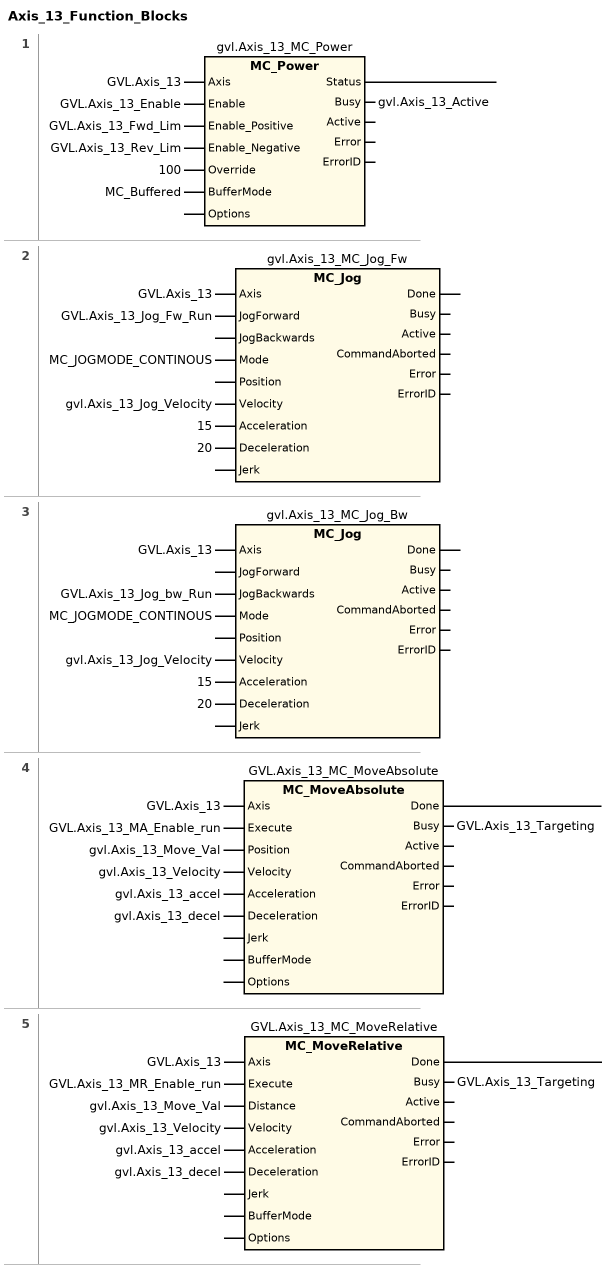
// NETWORK 1
gvl.Axis_13_MC_Power(
    Axis := GVL.Axis_13,
    Enable := GVL.Axis_13_Enable,
    Enable_Positive := GVL.Axis_13_Fwd_Lim,
    Enable_Negative := GVL.Axis_13_Rev_Lim,
    Override := 100,
    BufferMode := MC_Buffered,
    Busy => gvl.Axis_13_Active); // MC_Power

// NETWORK 2
gvl.Axis_13_MC_Jog_Fw(
    Axis := GVL.Axis_13,
    JogForward := GVL.Axis_13_Jog_Fw_Run,
    Mode := MC_JOGMODE_CONTINOUS,
    Velocity := gvl.Axis_13_Jog_Velocity,
    Acceleration := 15,
    Deceleration := 20); // MC_Jog

// NETWORK 3
gvl.Axis_13_MC_Jog_Bw(
    Axis := GVL.Axis_13,
    JogBackwards := GVL.Axis_13_Jog_bw_Run,
    Mode := MC_JOGMODE_CONTINOUS,
    Velocity := gvl.Axis_13_Jog_Velocity,
    Acceleration := 15,
    Deceleration := 20); // MC_Jog

// NETWORK 4
GVL.Axis_13_MC_MoveAbsolute(
    Axis := GVL.Axis_13,
    Execute := GVL.Axis_13_MA_Enable_run,
    Position := gvl.Axis_13_Move_Val,
    Velocity := gvl.Axis_13_Velocity,
    Acceleration := gvl.Axis_13_accel,
    Deceleration := gvl.Axis_13_decel,
    Busy => GVL.Axis_13_Targeting); // MC_MoveAbsolute

// NETWORK 5
GVL.Axis_13_MC_MoveRelative(
    Axis := GVL.Axis_13,
    Execute := GVL.Axis_13_MR_Enable_run,
    Distance := gvl.Axis_13_Move_Val,
    Velocity := gvl.Axis_13_Velocity,
    Acceleration := gvl.Axis_13_accel,
    Deceleration := gvl.Axis_13_decel,
    Busy => GVL.Axis_13_Targeting); // MC_MoveRelative

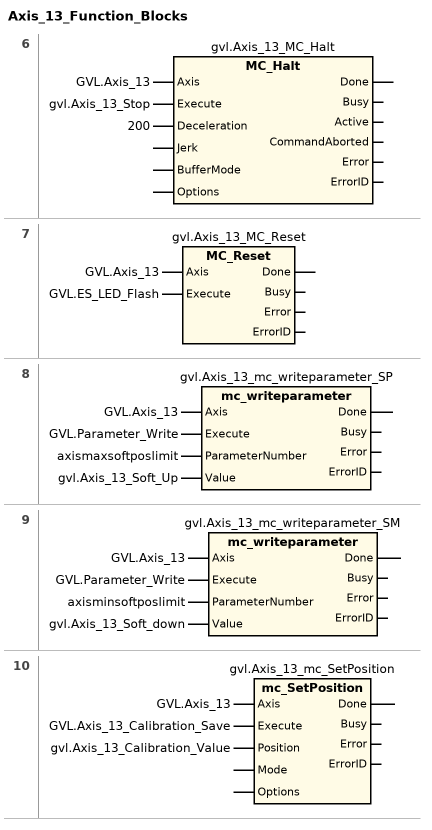
// NETWORK 6
gvl.Axis_13_MC_Halt(Axis := GVL.Axis_13, Execute := gvl.Axis_13_Stop, Deceleration := 200); // MC_Halt

// NETWORK 7
gvl.Axis_13_MC_Reset(Axis := GVL.Axis_13, Execute := GVL.ES_LED_Flash); // MC_Reset

// NETWORK 8
gvl.Axis_13_mc_writeparameter_SP(
    Axis := GVL.Axis_13,
    Execute := GVL.Parameter_Write,
    ParameterNumber := axismaxsoftposlimit,
    Value := gvl.Axis_13_Soft_Up); // mc_writeparameter

// NETWORK 9
gvl.Axis_13_mc_writeparameter_SM(
    Axis := GVL.Axis_13,
    Execute := GVL.Parameter_Write,
    ParameterNumber := axisminsoftposlimit,
    Value := gvl.Axis_13_Soft_down); // mc_writeparameter

// NETWORK 10
gvl.Axis_13_mc_SetPosition(
    Axis := GVL.Axis_13,
    Execute := GVL.Axis_13_Calibration_Save,
    Position := gvl.Axis_13_Calibration_Value); // mc_SetPosition

END_PROGRAM

// ---- POUs/Axis_13_Logic.TcPOU
PROGRAM Axis_13_Logic
VAR
	TON_0: TON;
	TON_1: TON;
	TON_2: TON;
	TON_3: TON;
	Axis_13_Velocity_Range: LREAL;
	Axis_13_Velocity_Scale: LREAL;
	Axis_13_Velocity_Raw: LREAL;
	Axis_13_Soft_Range: LREAL;
	Axis_13_Soft_Position: LREAL;
	Axis_13_Soft_Position_In_Range: LREAL;
END_VAR

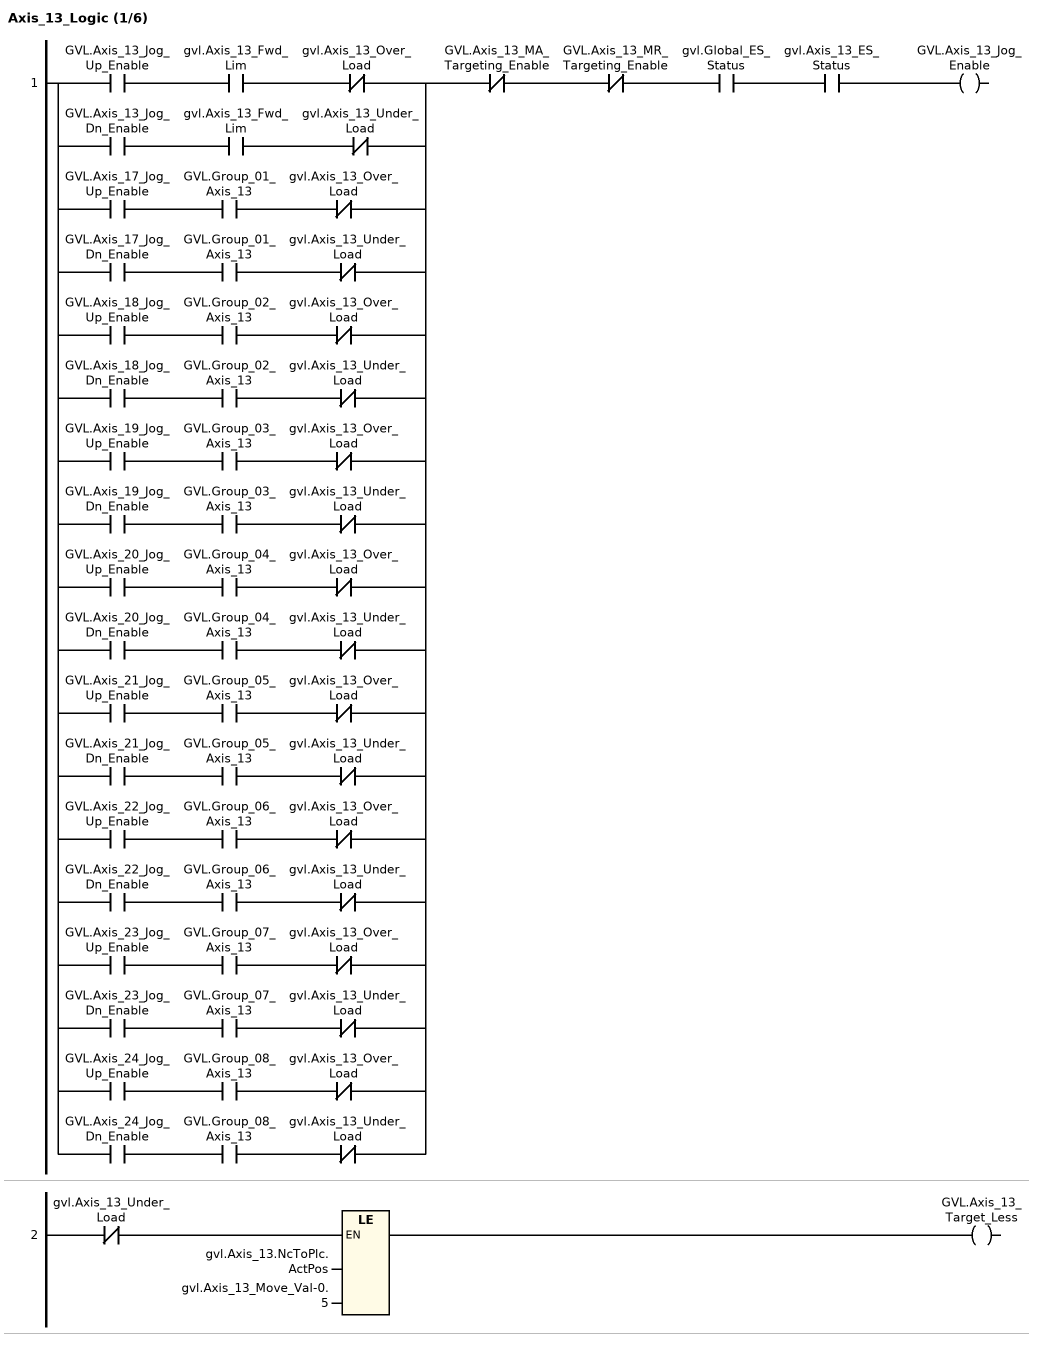
// NETWORK 1
GVL.Axis_13_Jog_Enable := (GVL.Axis_13_Jog_Up_Enable AND gvl.Axis_13_Fwd_Lim AND NOT gvl.Axis_13_Over_Load OR GVL.Axis_13_Jog_Dn_Enable AND gvl.Axis_13_Fwd_Lim AND NOT gvl.Axis_13_Under_Load OR GVL.Axis_17_Jog_Up_Enable AND GVL.Group_01_Axis_13 AND NOT gvl.Axis_13_Over_Load OR GVL.Axis_17_Jog_Dn_Enable AND GVL.Group_01_Axis_13 AND NOT gvl.Axis_13_Under_Load OR GVL.Axis_18_Jog_Up_Enable AND GVL.Group_02_Axis_13 AND NOT gvl.Axis_13_Over_Load OR GVL.Axis_18_Jog_Dn_Enable AND GVL.Group_02_Axis_13 AND NOT gvl.Axis_13_Under_Load OR GVL.Axis_19_Jog_Up_Enable AND GVL.Group_03_Axis_13 AND NOT gvl.Axis_13_Over_Load OR GVL.Axis_19_Jog_Dn_Enable AND GVL.Group_03_Axis_13 AND NOT gvl.Axis_13_Under_Load OR GVL.Axis_20_Jog_Up_Enable AND GVL.Group_04_Axis_13 AND NOT gvl.Axis_13_Over_Load OR GVL.Axis_20_Jog_Dn_Enable AND GVL.Group_04_Axis_13 AND NOT gvl.Axis_13_Under_Load OR GVL.Axis_21_Jog_Up_Enable AND GVL.Group_05_Axis_13 AND NOT gvl.Axis_13_Over_Load OR GVL.Axis_21_Jog_Dn_Enable AND GVL.Group_05_Axis_13 AND NOT gvl.Axis_13_Under_Load OR GVL.Axis_22_Jog_Up_Enable AND GVL.Group_06_Axis_13 AND NOT gvl.Axis_13_Over_Load OR GVL.Axis_22_Jog_Dn_Enable AND GVL.Group_06_Axis_13 AND NOT gvl.Axis_13_Under_Load OR GVL.Axis_23_Jog_Up_Enable AND GVL.Group_07_Axis_13 AND NOT gvl.Axis_13_Over_Load OR GVL.Axis_23_Jog_Dn_Enable AND GVL.Group_07_Axis_13 AND NOT gvl.Axis_13_Under_Load OR GVL.Axis_24_Jog_Up_Enable AND GVL.Group_08_Axis_13 AND NOT gvl.Axis_13_Over_Load OR GVL.Axis_24_Jog_Dn_Enable AND GVL.Group_08_Axis_13 AND NOT gvl.Axis_13_Under_Load) AND NOT GVL.Axis_13_MA_Targeting_Enable AND NOT GVL.Axis_13_MR_Targeting_Enable AND gvl.Global_ES_Status AND gvl.Axis_13_ES_Status;

// NETWORK 2
GVL.Axis_13_Target_Less := NOT gvl.Axis_13_Under_Load AND gvl.Axis_13.NcToPlc.ActPos <= (gvl.Axis_13_Move_Val-0.5);

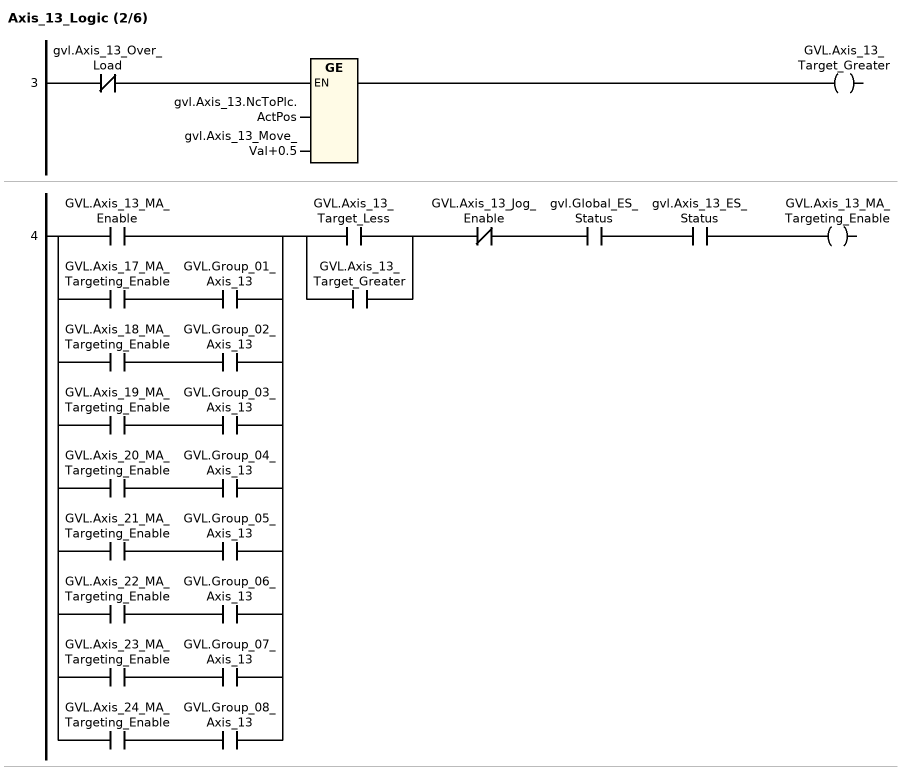
// NETWORK 3
GVL.Axis_13_Target_Greater := NOT gvl.Axis_13_Over_Load AND gvl.Axis_13.NcToPlc.ActPos >= (gvl.Axis_13_Move_Val+0.5);

// NETWORK 4
GVL.Axis_13_MA_Targeting_Enable := (GVL.Axis_13_MA_Enable OR GVL.Axis_17_MA_Targeting_Enable AND GVL.Group_01_Axis_13 OR GVL.Axis_18_MA_Targeting_Enable AND GVL.Group_02_Axis_13 OR GVL.Axis_19_MA_Targeting_Enable AND GVL.Group_03_Axis_13 OR GVL.Axis_20_MA_Targeting_Enable AND GVL.Group_04_Axis_13 OR GVL.Axis_21_MA_Targeting_Enable AND GVL.Group_05_Axis_13 OR GVL.Axis_22_MA_Targeting_Enable AND GVL.Group_06_Axis_13 OR GVL.Axis_23_MA_Targeting_Enable AND GVL.Group_07_Axis_13 OR GVL.Axis_24_MA_Targeting_Enable AND GVL.Group_08_Axis_13) AND (GVL.Axis_13_Target_Less OR GVL.Axis_13_Target_Greater) AND NOT GVL.Axis_13_Jog_Enable AND gvl.Global_ES_Status AND gvl.Axis_13_ES_Status;

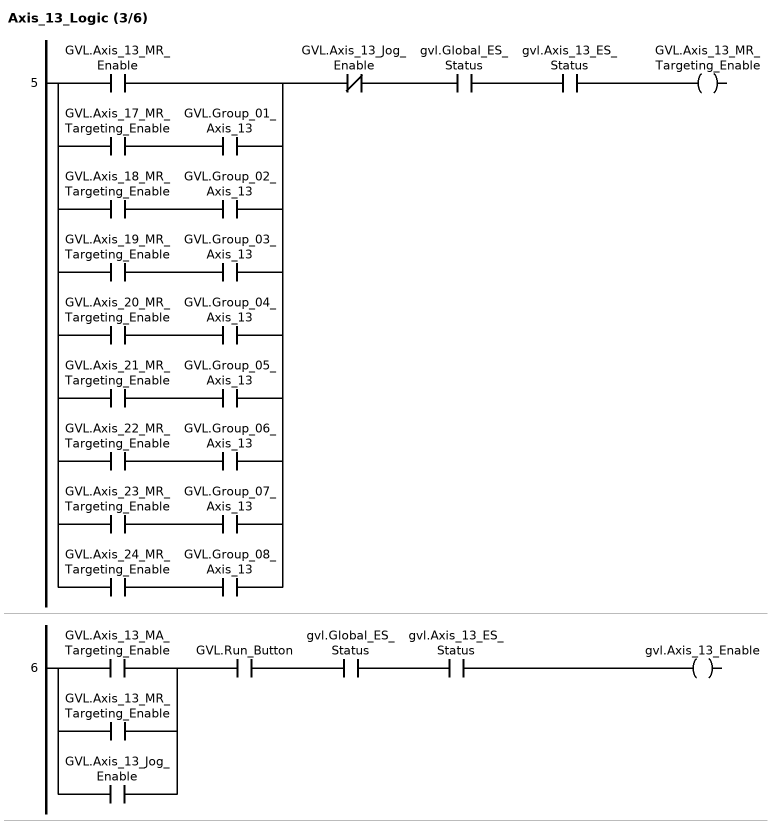
// NETWORK 5
GVL.Axis_13_MR_Targeting_Enable := (GVL.Axis_13_MR_Enable OR GVL.Axis_17_MR_Targeting_Enable AND GVL.Group_01_Axis_13 OR GVL.Axis_18_MR_Targeting_Enable AND GVL.Group_02_Axis_13 OR GVL.Axis_19_MR_Targeting_Enable AND GVL.Group_03_Axis_13 OR GVL.Axis_20_MR_Targeting_Enable AND GVL.Group_04_Axis_13 OR GVL.Axis_21_MR_Targeting_Enable AND GVL.Group_05_Axis_13 OR GVL.Axis_22_MR_Targeting_Enable AND GVL.Group_06_Axis_13 OR GVL.Axis_23_MR_Targeting_Enable AND GVL.Group_07_Axis_13 OR GVL.Axis_24_MR_Targeting_Enable AND GVL.Group_08_Axis_13) AND NOT GVL.Axis_13_Jog_Enable AND gvl.Global_ES_Status AND gvl.Axis_13_ES_Status;

// NETWORK 6
gvl.Axis_13_Enable := (GVL.Axis_13_MA_Targeting_Enable OR GVL.Axis_13_MR_Targeting_Enable OR GVL.Axis_13_Jog_Enable) AND GVL.Run_Button AND gvl.Global_ES_Status AND gvl.Axis_13_ES_Status;

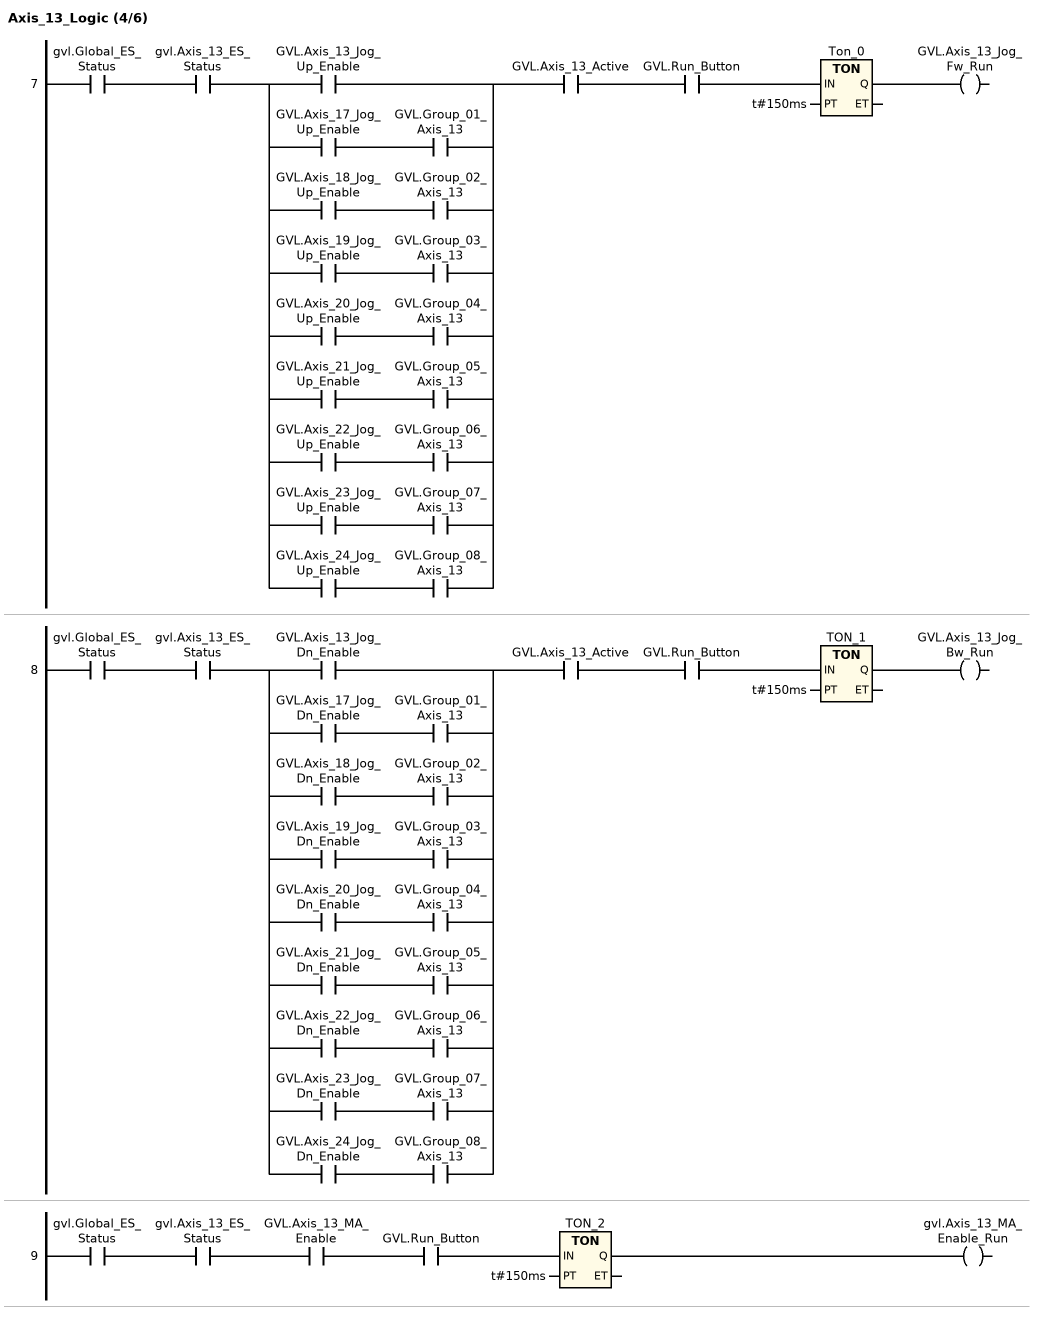
// NETWORK 7
Ton_0(IN := gvl.Global_ES_Status AND gvl.Axis_13_ES_Status AND (GVL.Axis_13_Jog_Up_Enable OR GVL.Axis_17_Jog_Up_Enable AND GVL.Group_01_Axis_13 OR GVL.Axis_18_Jog_Up_Enable AND GVL.Group_02_Axis_13 OR GVL.Axis_19_Jog_Up_Enable AND GVL.Group_03_Axis_13 OR GVL.Axis_20_Jog_Up_Enable AND GVL.Group_04_Axis_13 OR GVL.Axis_21_Jog_Up_Enable AND GVL.Group_05_Axis_13 OR GVL.Axis_22_Jog_Up_Enable AND GVL.Group_06_Axis_13 OR GVL.Axis_23_Jog_Up_Enable AND GVL.Group_07_Axis_13 OR GVL.Axis_24_Jog_Up_Enable AND GVL.Group_08_Axis_13) AND GVL.Axis_13_Active AND GVL.Run_Button, PT := t#150ms); // TON
GVL.Axis_13_Jog_Fw_Run := Ton_0.Q;

// NETWORK 8
TON_1(IN := gvl.Global_ES_Status AND gvl.Axis_13_ES_Status AND (GVL.Axis_13_Jog_Dn_Enable OR GVL.Axis_17_Jog_Dn_Enable AND GVL.Group_01_Axis_13 OR GVL.Axis_18_Jog_Dn_Enable AND GVL.Group_02_Axis_13 OR GVL.Axis_19_Jog_Dn_Enable AND GVL.Group_03_Axis_13 OR GVL.Axis_20_Jog_Dn_Enable AND GVL.Group_04_Axis_13 OR GVL.Axis_21_Jog_Dn_Enable AND GVL.Group_05_Axis_13 OR GVL.Axis_22_Jog_Dn_Enable AND GVL.Group_06_Axis_13 OR GVL.Axis_23_Jog_Dn_Enable AND GVL.Group_07_Axis_13 OR GVL.Axis_24_Jog_Dn_Enable AND GVL.Group_08_Axis_13) AND GVL.Axis_13_Active AND GVL.Run_Button, PT := t#150ms); // TON
GVL.Axis_13_Jog_Bw_Run := TON_1.Q;

// NETWORK 9
TON_2(IN := gvl.Global_ES_Status AND gvl.Axis_13_ES_Status AND GVL.Axis_13_MA_Enable AND GVL.Run_Button, PT := t#150ms); // TON
gvl.Axis_13_MA_Enable_Run := TON_2.Q;

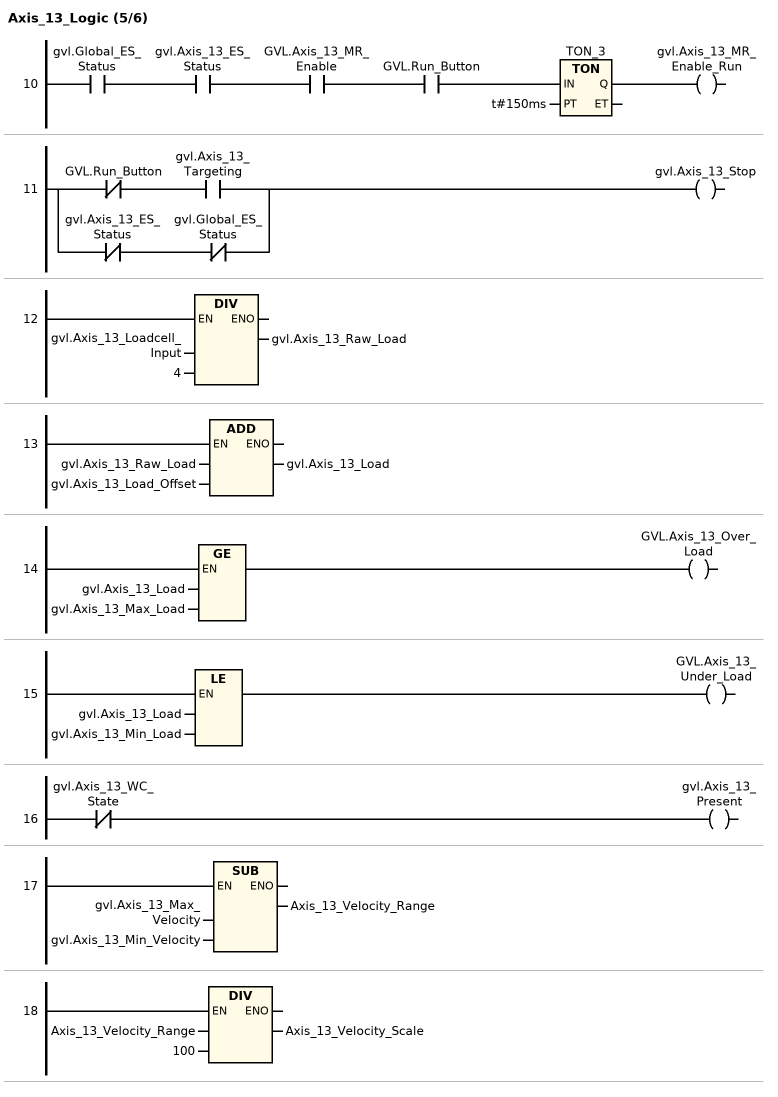
// NETWORK 10
TON_3(IN := gvl.Global_ES_Status AND gvl.Axis_13_ES_Status AND GVL.Axis_13_MR_Enable AND GVL.Run_Button, PT := t#150ms); // TON
gvl.Axis_13_MR_Enable_Run := TON_3.Q;

// NETWORK 11
gvl.Axis_13_Stop := NOT GVL.Run_Button AND gvl.Axis_13_Targeting OR NOT gvl.Axis_13_ES_Status AND NOT gvl.Global_ES_Status;

// NETWORK 12
gvl.Axis_13_Raw_Load := gvl.Axis_13_Loadcell_Input / 4;

// NETWORK 13
gvl.Axis_13_Load := gvl.Axis_13_Raw_Load + gvl.Axis_13_Load_Offset;

// NETWORK 14
GVL.Axis_13_Over_Load := gvl.Axis_13_Load >= gvl.Axis_13_Max_Load;

// NETWORK 15
GVL.Axis_13_Under_Load := gvl.Axis_13_Load <= gvl.Axis_13_Min_Load;

// NETWORK 16
gvl.Axis_13_Present := NOT gvl.Axis_13_WC_State;

// NETWORK 17
Axis_13_Velocity_Range := gvl.Axis_13_Max_Velocity - gvl.Axis_13_Min_Velocity;

// NETWORK 18
Axis_13_Velocity_Scale := Axis_13_Velocity_Range / 100;

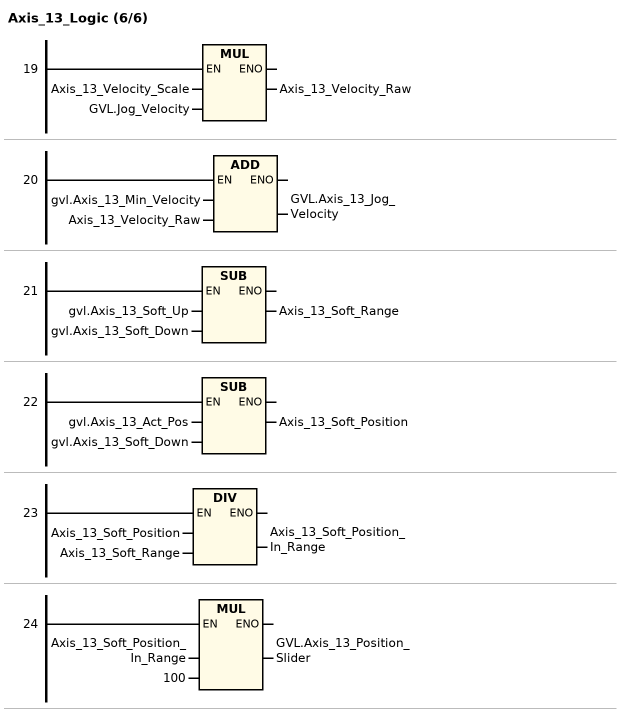
// NETWORK 19
Axis_13_Velocity_Raw := Axis_13_Velocity_Scale * GVL.Jog_Velocity;

// NETWORK 20
GVL.Axis_13_Jog_Velocity := gvl.Axis_13_Min_Velocity + Axis_13_Velocity_Raw;

// NETWORK 21
Axis_13_Soft_Range := gvl.Axis_13_Soft_Up - gvl.Axis_13_Soft_Down;

// NETWORK 22
Axis_13_Soft_Position := gvl.Axis_13_Act_Pos - gvl.Axis_13_Soft_Down;

// NETWORK 23
Axis_13_Soft_Position_In_Range := Axis_13_Soft_Position / Axis_13_Soft_Range;

// NETWORK 24
GVL.Axis_13_Position_Slider := Axis_13_Soft_Position_In_Range * 100;

END_PROGRAM

// ---- POUs/Axis_14_Function_Blocks.TcPOU
PROGRAM Axis_14_Function_Blocks
VAR
END_VAR

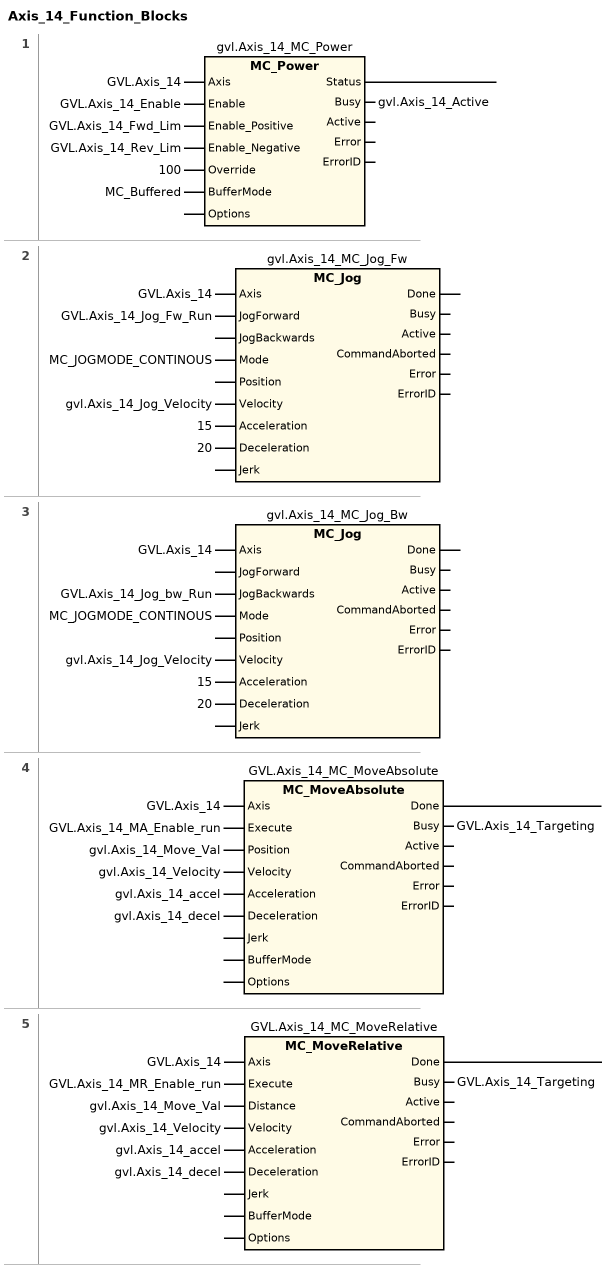
// NETWORK 1
gvl.Axis_14_MC_Power(
    Axis := GVL.Axis_14,
    Enable := GVL.Axis_14_Enable,
    Enable_Positive := GVL.Axis_14_Fwd_Lim,
    Enable_Negative := GVL.Axis_14_Rev_Lim,
    Override := 100,
    BufferMode := MC_Buffered,
    Busy => gvl.Axis_14_Active); // MC_Power

// NETWORK 2
gvl.Axis_14_MC_Jog_Fw(
    Axis := GVL.Axis_14,
    JogForward := GVL.Axis_14_Jog_Fw_Run,
    Mode := MC_JOGMODE_CONTINOUS,
    Velocity := gvl.Axis_14_Jog_Velocity,
    Acceleration := 15,
    Deceleration := 20); // MC_Jog

// NETWORK 3
gvl.Axis_14_MC_Jog_Bw(
    Axis := GVL.Axis_14,
    JogBackwards := GVL.Axis_14_Jog_bw_Run,
    Mode := MC_JOGMODE_CONTINOUS,
    Velocity := gvl.Axis_14_Jog_Velocity,
    Acceleration := 15,
    Deceleration := 20); // MC_Jog

// NETWORK 4
GVL.Axis_14_MC_MoveAbsolute(
    Axis := GVL.Axis_14,
    Execute := GVL.Axis_14_MA_Enable_run,
    Position := gvl.Axis_14_Move_Val,
    Velocity := gvl.Axis_14_Velocity,
    Acceleration := gvl.Axis_14_accel,
    Deceleration := gvl.Axis_14_decel,
    Busy => GVL.Axis_14_Targeting); // MC_MoveAbsolute

// NETWORK 5
GVL.Axis_14_MC_MoveRelative(
    Axis := GVL.Axis_14,
    Execute := GVL.Axis_14_MR_Enable_run,
    Distance := gvl.Axis_14_Move_Val,
    Velocity := gvl.Axis_14_Velocity,
    Acceleration := gvl.Axis_14_accel,
    Deceleration := gvl.Axis_14_decel,
    Busy => GVL.Axis_14_Targeting); // MC_MoveRelative

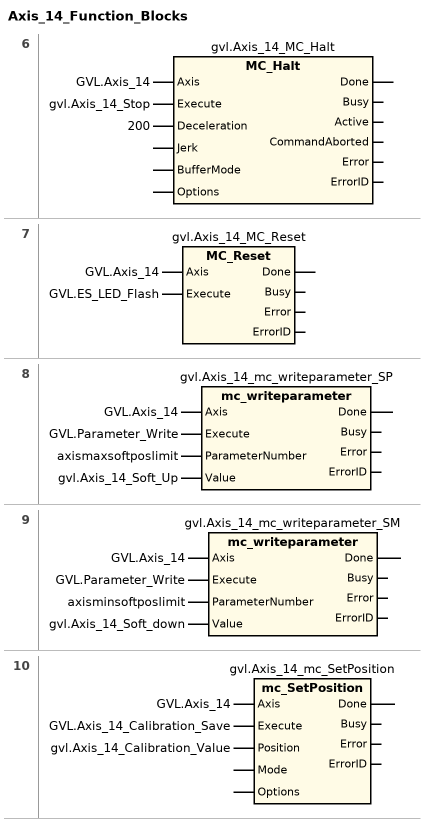
// NETWORK 6
gvl.Axis_14_MC_Halt(Axis := GVL.Axis_14, Execute := gvl.Axis_14_Stop, Deceleration := 200); // MC_Halt

// NETWORK 7
gvl.Axis_14_MC_Reset(Axis := GVL.Axis_14, Execute := GVL.ES_LED_Flash); // MC_Reset

// NETWORK 8
gvl.Axis_14_mc_writeparameter_SP(
    Axis := GVL.Axis_14,
    Execute := GVL.Parameter_Write,
    ParameterNumber := axismaxsoftposlimit,
    Value := gvl.Axis_14_Soft_Up); // mc_writeparameter

// NETWORK 9
gvl.Axis_14_mc_writeparameter_SM(
    Axis := GVL.Axis_14,
    Execute := GVL.Parameter_Write,
    ParameterNumber := axisminsoftposlimit,
    Value := gvl.Axis_14_Soft_down); // mc_writeparameter

// NETWORK 10
gvl.Axis_14_mc_SetPosition(
    Axis := GVL.Axis_14,
    Execute := GVL.Axis_14_Calibration_Save,
    Position := gvl.Axis_14_Calibration_Value); // mc_SetPosition

END_PROGRAM

// ---- POUs/Axis_14_Logic.TcPOU
PROGRAM Axis_14_Logic
VAR
	TON_0: TON;
	TON_1: TON;
	TON_2: TON;
	TON_3: TON;
	Axis_14_Velocity_Range: LREAL;
	Axis_14_Velocity_Scale: LREAL;
	Axis_14_Velocity_Raw: LREAL;
	Axis_14_Soft_Range: LREAL;
	Axis_14_Soft_Position: LREAL;
	Axis_14_Soft_Position_In_Range: LREAL;
END_VAR

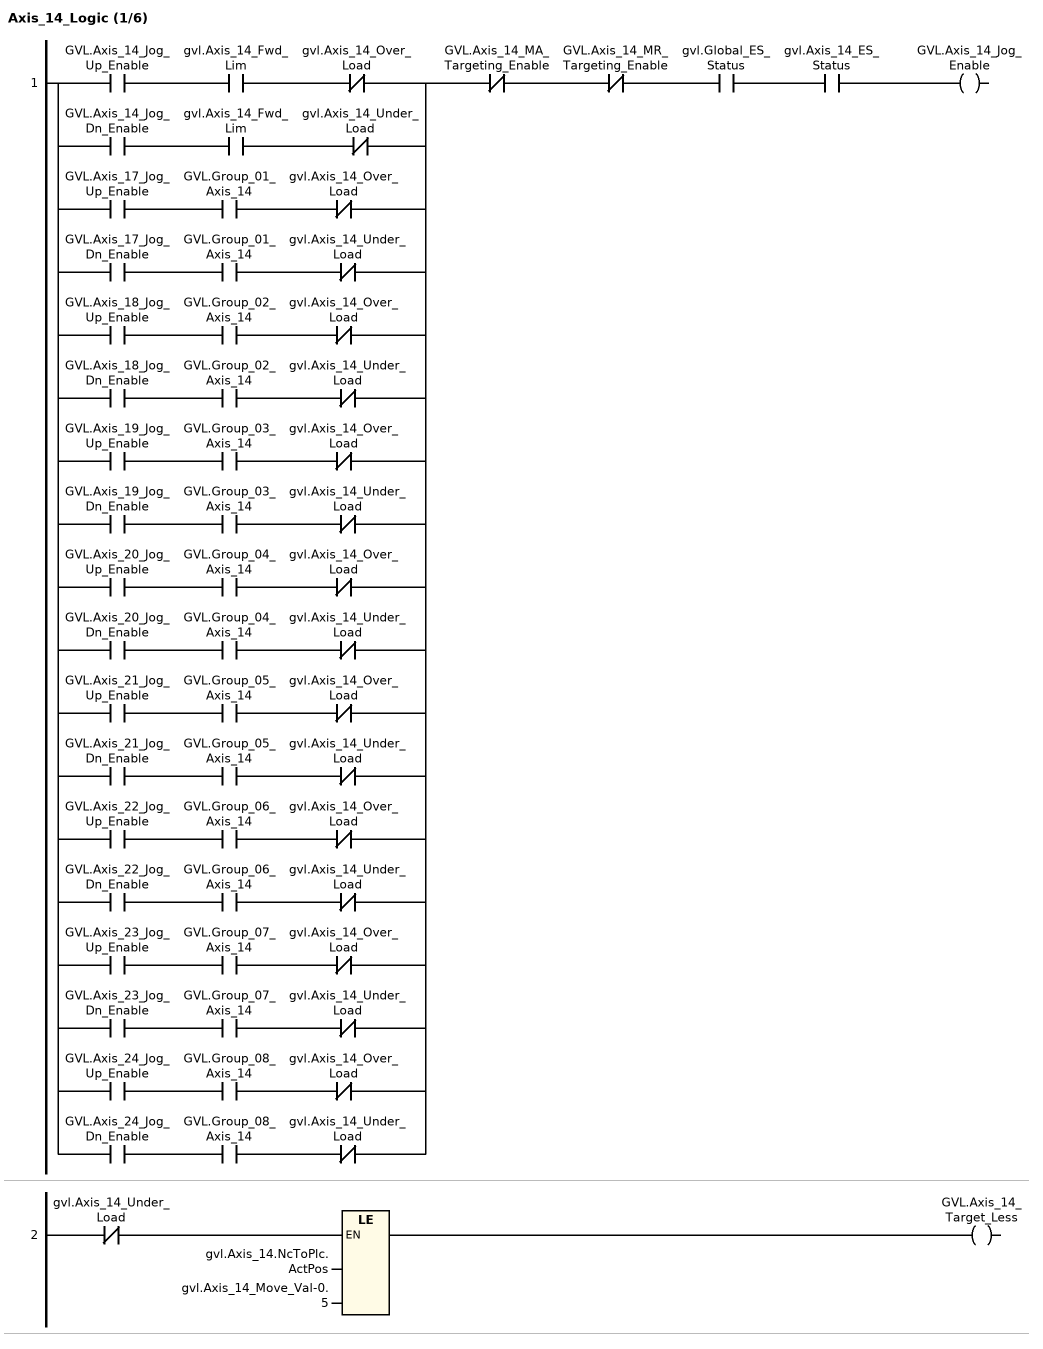
// NETWORK 1
GVL.Axis_14_Jog_Enable := (GVL.Axis_14_Jog_Up_Enable AND gvl.Axis_14_Fwd_Lim AND NOT gvl.Axis_14_Over_Load OR GVL.Axis_14_Jog_Dn_Enable AND gvl.Axis_14_Fwd_Lim AND NOT gvl.Axis_14_Under_Load OR GVL.Axis_17_Jog_Up_Enable AND GVL.Group_01_Axis_14 AND NOT gvl.Axis_14_Over_Load OR GVL.Axis_17_Jog_Dn_Enable AND GVL.Group_01_Axis_14 AND NOT gvl.Axis_14_Under_Load OR GVL.Axis_18_Jog_Up_Enable AND GVL.Group_02_Axis_14 AND NOT gvl.Axis_14_Over_Load OR GVL.Axis_18_Jog_Dn_Enable AND GVL.Group_02_Axis_14 AND NOT gvl.Axis_14_Under_Load OR GVL.Axis_19_Jog_Up_Enable AND GVL.Group_03_Axis_14 AND NOT gvl.Axis_14_Over_Load OR GVL.Axis_19_Jog_Dn_Enable AND GVL.Group_03_Axis_14 AND NOT gvl.Axis_14_Under_Load OR GVL.Axis_20_Jog_Up_Enable AND GVL.Group_04_Axis_14 AND NOT gvl.Axis_14_Over_Load OR GVL.Axis_20_Jog_Dn_Enable AND GVL.Group_04_Axis_14 AND NOT gvl.Axis_14_Under_Load OR GVL.Axis_21_Jog_Up_Enable AND GVL.Group_05_Axis_14 AND NOT gvl.Axis_14_Over_Load OR GVL.Axis_21_Jog_Dn_Enable AND GVL.Group_05_Axis_14 AND NOT gvl.Axis_14_Under_Load OR GVL.Axis_22_Jog_Up_Enable AND GVL.Group_06_Axis_14 AND NOT gvl.Axis_14_Over_Load OR GVL.Axis_22_Jog_Dn_Enable AND GVL.Group_06_Axis_14 AND NOT gvl.Axis_14_Under_Load OR GVL.Axis_23_Jog_Up_Enable AND GVL.Group_07_Axis_14 AND NOT gvl.Axis_14_Over_Load OR GVL.Axis_23_Jog_Dn_Enable AND GVL.Group_07_Axis_14 AND NOT gvl.Axis_14_Under_Load OR GVL.Axis_24_Jog_Up_Enable AND GVL.Group_08_Axis_14 AND NOT gvl.Axis_14_Over_Load OR GVL.Axis_24_Jog_Dn_Enable AND GVL.Group_08_Axis_14 AND NOT gvl.Axis_14_Under_Load) AND NOT GVL.Axis_14_MA_Targeting_Enable AND NOT GVL.Axis_14_MR_Targeting_Enable AND gvl.Global_ES_Status AND gvl.Axis_14_ES_Status;

// NETWORK 2
GVL.Axis_14_Target_Less := NOT gvl.Axis_14_Under_Load AND gvl.Axis_14.NcToPlc.ActPos <= (gvl.Axis_14_Move_Val-0.5);

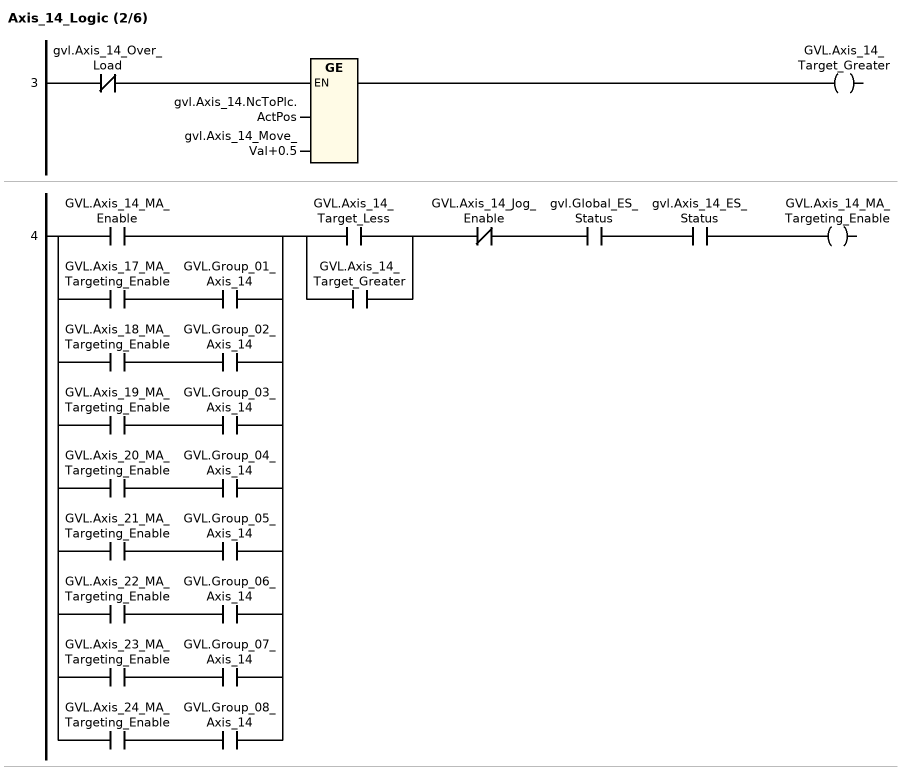
// NETWORK 3
GVL.Axis_14_Target_Greater := NOT gvl.Axis_14_Over_Load AND gvl.Axis_14.NcToPlc.ActPos >= (gvl.Axis_14_Move_Val+0.5);

// NETWORK 4
GVL.Axis_14_MA_Targeting_Enable := (GVL.Axis_14_MA_Enable OR GVL.Axis_17_MA_Targeting_Enable AND GVL.Group_01_Axis_14 OR GVL.Axis_18_MA_Targeting_Enable AND GVL.Group_02_Axis_14 OR GVL.Axis_19_MA_Targeting_Enable AND GVL.Group_03_Axis_14 OR GVL.Axis_20_MA_Targeting_Enable AND GVL.Group_04_Axis_14 OR GVL.Axis_21_MA_Targeting_Enable AND GVL.Group_05_Axis_14 OR GVL.Axis_22_MA_Targeting_Enable AND GVL.Group_06_Axis_14 OR GVL.Axis_23_MA_Targeting_Enable AND GVL.Group_07_Axis_14 OR GVL.Axis_24_MA_Targeting_Enable AND GVL.Group_08_Axis_14) AND (GVL.Axis_14_Target_Less OR GVL.Axis_14_Target_Greater) AND NOT GVL.Axis_14_Jog_Enable AND gvl.Global_ES_Status AND gvl.Axis_14_ES_Status;

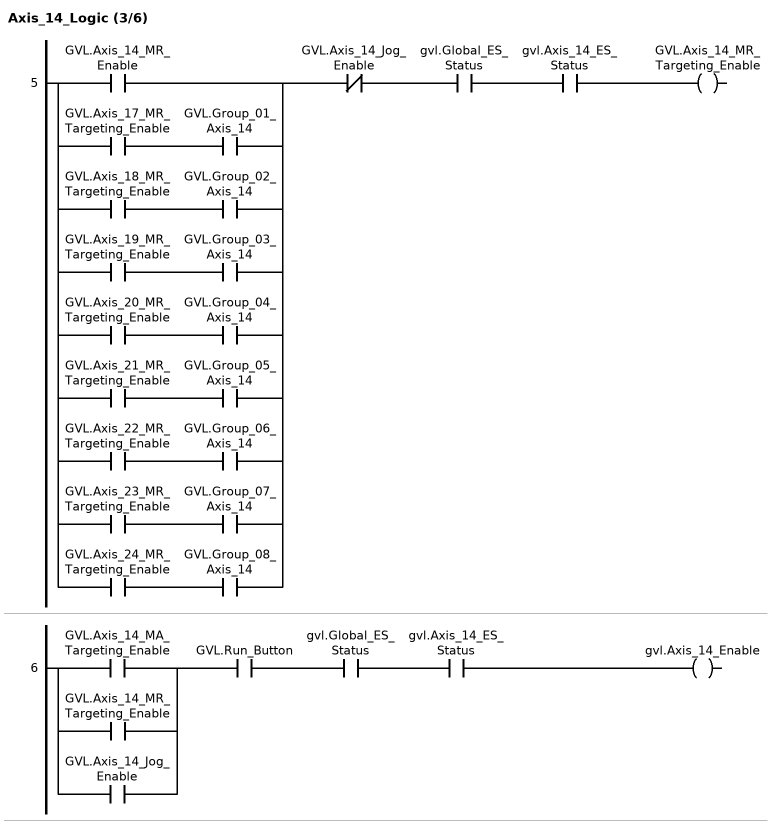
// NETWORK 5
GVL.Axis_14_MR_Targeting_Enable := (GVL.Axis_14_MR_Enable OR GVL.Axis_17_MR_Targeting_Enable AND GVL.Group_01_Axis_14 OR GVL.Axis_18_MR_Targeting_Enable AND GVL.Group_02_Axis_14 OR GVL.Axis_19_MR_Targeting_Enable AND GVL.Group_03_Axis_14 OR GVL.Axis_20_MR_Targeting_Enable AND GVL.Group_04_Axis_14 OR GVL.Axis_21_MR_Targeting_Enable AND GVL.Group_05_Axis_14 OR GVL.Axis_22_MR_Targeting_Enable AND GVL.Group_06_Axis_14 OR GVL.Axis_23_MR_Targeting_Enable AND GVL.Group_07_Axis_14 OR GVL.Axis_24_MR_Targeting_Enable AND GVL.Group_08_Axis_14) AND NOT GVL.Axis_14_Jog_Enable AND gvl.Global_ES_Status AND gvl.Axis_14_ES_Status;

// NETWORK 6
gvl.Axis_14_Enable := (GVL.Axis_14_MA_Targeting_Enable OR GVL.Axis_14_MR_Targeting_Enable OR GVL.Axis_14_Jog_Enable) AND GVL.Run_Button AND gvl.Global_ES_Status AND gvl.Axis_14_ES_Status;

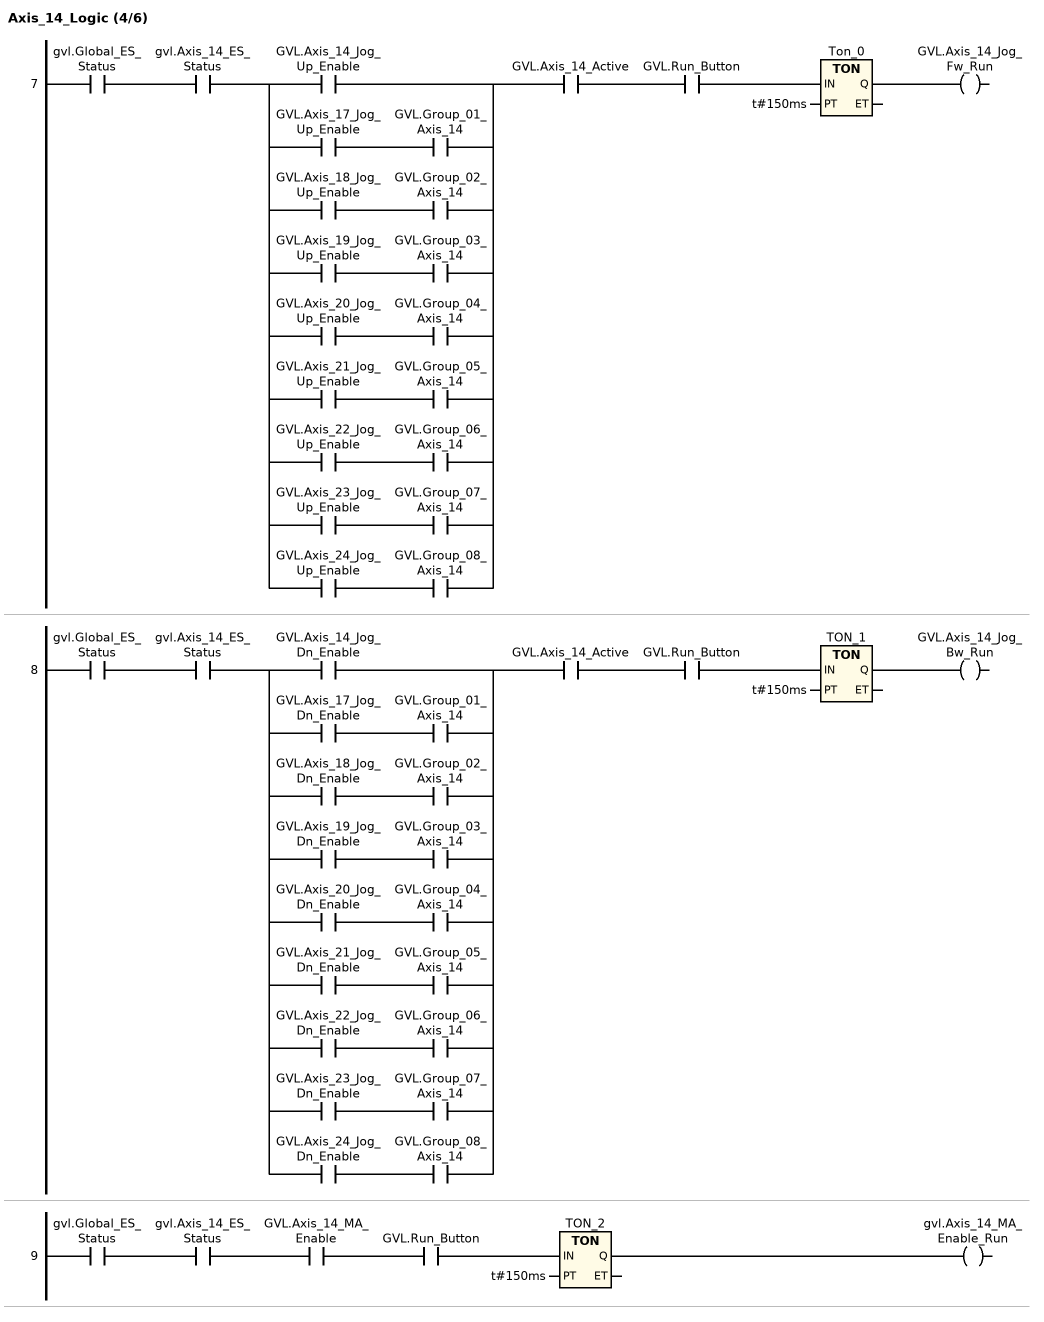
// NETWORK 7
Ton_0(IN := gvl.Global_ES_Status AND gvl.Axis_14_ES_Status AND (GVL.Axis_14_Jog_Up_Enable OR GVL.Axis_17_Jog_Up_Enable AND GVL.Group_01_Axis_14 OR GVL.Axis_18_Jog_Up_Enable AND GVL.Group_02_Axis_14 OR GVL.Axis_19_Jog_Up_Enable AND GVL.Group_03_Axis_14 OR GVL.Axis_20_Jog_Up_Enable AND GVL.Group_04_Axis_14 OR GVL.Axis_21_Jog_Up_Enable AND GVL.Group_05_Axis_14 OR GVL.Axis_22_Jog_Up_Enable AND GVL.Group_06_Axis_14 OR GVL.Axis_23_Jog_Up_Enable AND GVL.Group_07_Axis_14 OR GVL.Axis_24_Jog_Up_Enable AND GVL.Group_08_Axis_14) AND GVL.Axis_14_Active AND GVL.Run_Button, PT := t#150ms); // TON
GVL.Axis_14_Jog_Fw_Run := Ton_0.Q;

// NETWORK 8
TON_1(IN := gvl.Global_ES_Status AND gvl.Axis_14_ES_Status AND (GVL.Axis_14_Jog_Dn_Enable OR GVL.Axis_17_Jog_Dn_Enable AND GVL.Group_01_Axis_14 OR GVL.Axis_18_Jog_Dn_Enable AND GVL.Group_02_Axis_14 OR GVL.Axis_19_Jog_Dn_Enable AND GVL.Group_03_Axis_14 OR GVL.Axis_20_Jog_Dn_Enable AND GVL.Group_04_Axis_14 OR GVL.Axis_21_Jog_Dn_Enable AND GVL.Group_05_Axis_14 OR GVL.Axis_22_Jog_Dn_Enable AND GVL.Group_06_Axis_14 OR GVL.Axis_23_Jog_Dn_Enable AND GVL.Group_07_Axis_14 OR GVL.Axis_24_Jog_Dn_Enable AND GVL.Group_08_Axis_14) AND GVL.Axis_14_Active AND GVL.Run_Button, PT := t#150ms); // TON
GVL.Axis_14_Jog_Bw_Run := TON_1.Q;

// NETWORK 9
TON_2(IN := gvl.Global_ES_Status AND gvl.Axis_14_ES_Status AND GVL.Axis_14_MA_Enable AND GVL.Run_Button, PT := t#150ms); // TON
gvl.Axis_14_MA_Enable_Run := TON_2.Q;

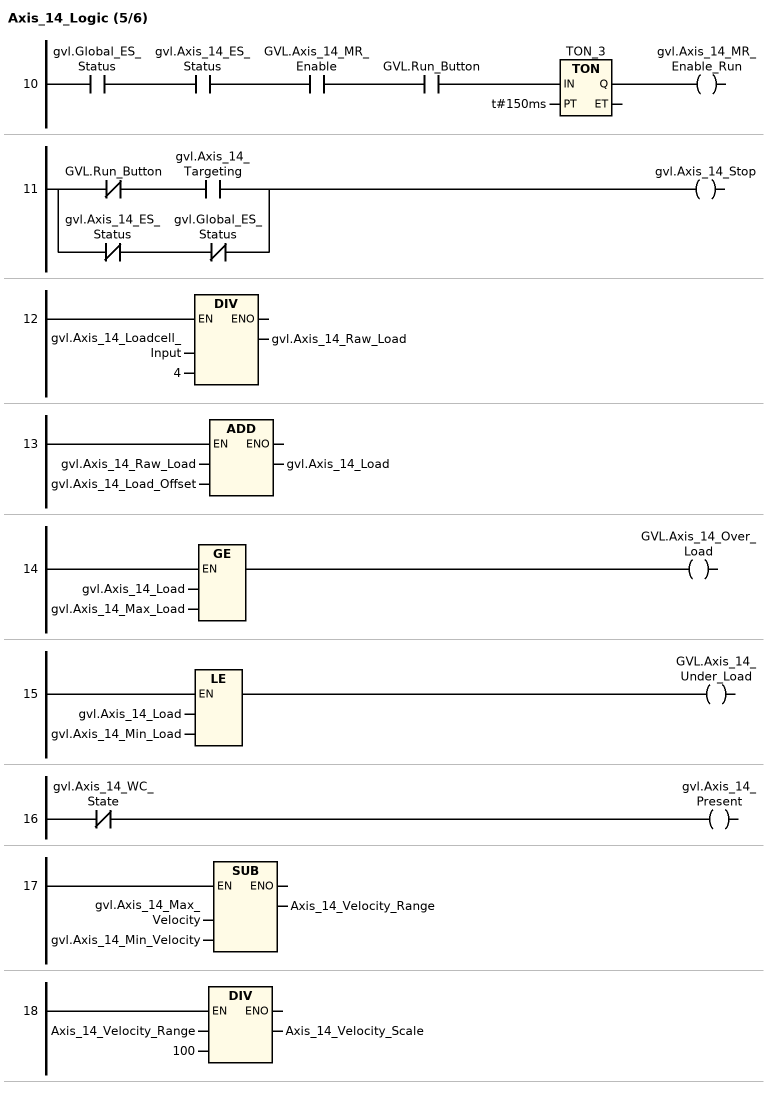
// NETWORK 10
TON_3(IN := gvl.Global_ES_Status AND gvl.Axis_14_ES_Status AND GVL.Axis_14_MR_Enable AND GVL.Run_Button, PT := t#150ms); // TON
gvl.Axis_14_MR_Enable_Run := TON_3.Q;

// NETWORK 11
gvl.Axis_14_Stop := NOT GVL.Run_Button AND gvl.Axis_14_Targeting OR NOT gvl.Axis_14_ES_Status AND NOT gvl.Global_ES_Status;

// NETWORK 12
gvl.Axis_14_Raw_Load := gvl.Axis_14_Loadcell_Input / 4;

// NETWORK 13
gvl.Axis_14_Load := gvl.Axis_14_Raw_Load + gvl.Axis_14_Load_Offset;

// NETWORK 14
GVL.Axis_14_Over_Load := gvl.Axis_14_Load >= gvl.Axis_14_Max_Load;

// NETWORK 15
GVL.Axis_14_Under_Load := gvl.Axis_14_Load <= gvl.Axis_14_Min_Load;

// NETWORK 16
gvl.Axis_14_Present := NOT gvl.Axis_14_WC_State;

// NETWORK 17
Axis_14_Velocity_Range := gvl.Axis_14_Max_Velocity - gvl.Axis_14_Min_Velocity;

// NETWORK 18
Axis_14_Velocity_Scale := Axis_14_Velocity_Range / 100;

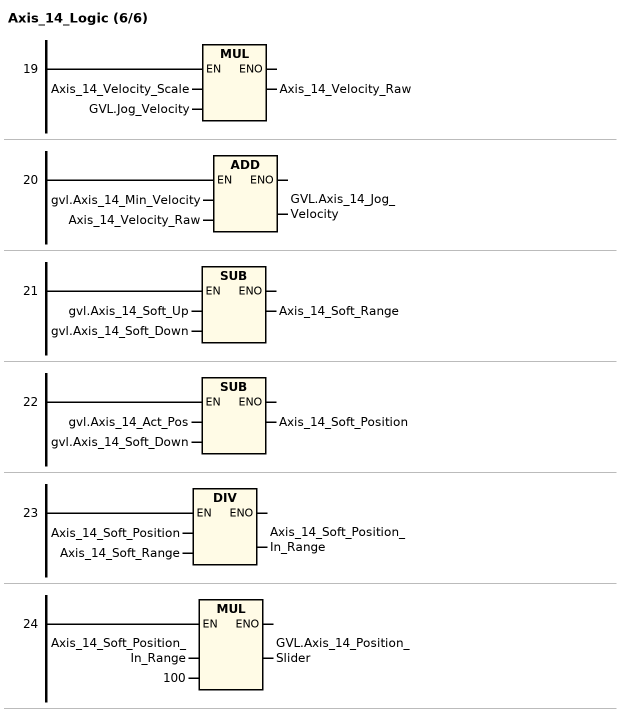
// NETWORK 19
Axis_14_Velocity_Raw := Axis_14_Velocity_Scale * GVL.Jog_Velocity;

// NETWORK 20
GVL.Axis_14_Jog_Velocity := gvl.Axis_14_Min_Velocity + Axis_14_Velocity_Raw;

// NETWORK 21
Axis_14_Soft_Range := gvl.Axis_14_Soft_Up - gvl.Axis_14_Soft_Down;

// NETWORK 22
Axis_14_Soft_Position := gvl.Axis_14_Act_Pos - gvl.Axis_14_Soft_Down;

// NETWORK 23
Axis_14_Soft_Position_In_Range := Axis_14_Soft_Position / Axis_14_Soft_Range;

// NETWORK 24
GVL.Axis_14_Position_Slider := Axis_14_Soft_Position_In_Range * 100;

END_PROGRAM

// ---- POUs/Axis_15_Function_Blocks.TcPOU
PROGRAM Axis_15_Function_Blocks
VAR
END_VAR

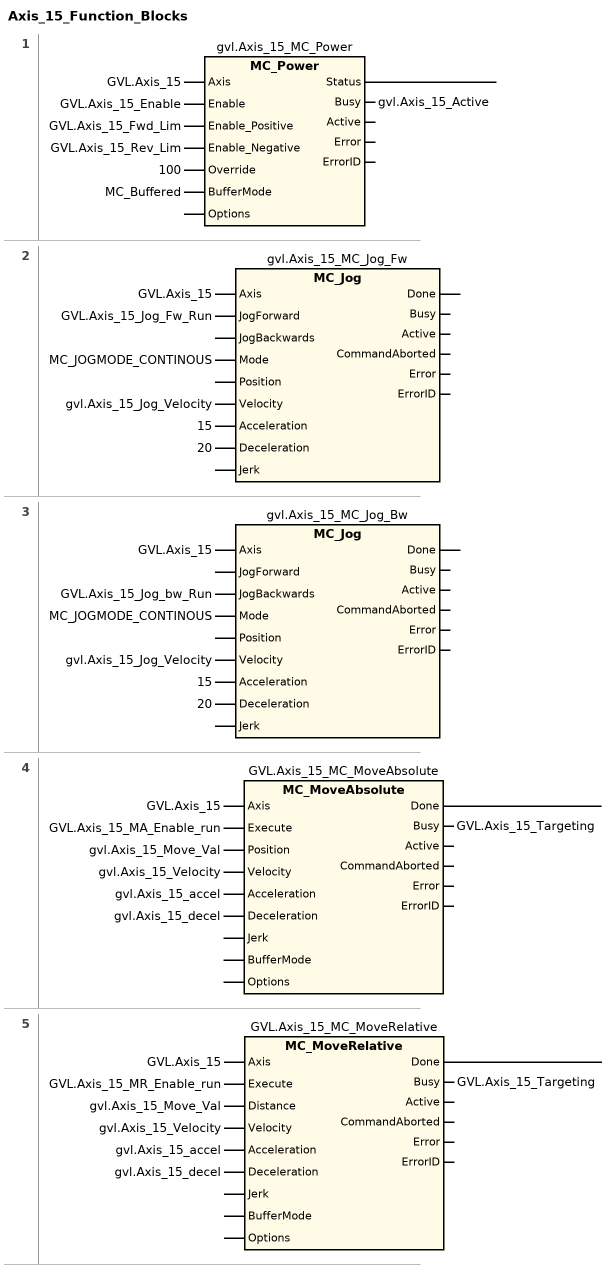
// NETWORK 1
gvl.Axis_15_MC_Power(
    Axis := GVL.Axis_15,
    Enable := GVL.Axis_15_Enable,
    Enable_Positive := GVL.Axis_15_Fwd_Lim,
    Enable_Negative := GVL.Axis_15_Rev_Lim,
    Override := 100,
    BufferMode := MC_Buffered,
    Busy => gvl.Axis_15_Active); // MC_Power

// NETWORK 2
gvl.Axis_15_MC_Jog_Fw(
    Axis := GVL.Axis_15,
    JogForward := GVL.Axis_15_Jog_Fw_Run,
    Mode := MC_JOGMODE_CONTINOUS,
    Velocity := gvl.Axis_15_Jog_Velocity,
    Acceleration := 15,
    Deceleration := 20); // MC_Jog

// NETWORK 3
gvl.Axis_15_MC_Jog_Bw(
    Axis := GVL.Axis_15,
    JogBackwards := GVL.Axis_15_Jog_bw_Run,
    Mode := MC_JOGMODE_CONTINOUS,
    Velocity := gvl.Axis_15_Jog_Velocity,
    Acceleration := 15,
    Deceleration := 20); // MC_Jog

// NETWORK 4
GVL.Axis_15_MC_MoveAbsolute(
    Axis := GVL.Axis_15,
    Execute := GVL.Axis_15_MA_Enable_run,
    Position := gvl.Axis_15_Move_Val,
    Velocity := gvl.Axis_15_Velocity,
    Acceleration := gvl.Axis_15_accel,
    Deceleration := gvl.Axis_15_decel,
    Busy => GVL.Axis_15_Targeting); // MC_MoveAbsolute

// NETWORK 5
GVL.Axis_15_MC_MoveRelative(
    Axis := GVL.Axis_15,
    Execute := GVL.Axis_15_MR_Enable_run,
    Distance := gvl.Axis_15_Move_Val,
    Velocity := gvl.Axis_15_Velocity,
    Acceleration := gvl.Axis_15_accel,
    Deceleration := gvl.Axis_15_decel,
    Busy => GVL.Axis_15_Targeting); // MC_MoveRelative

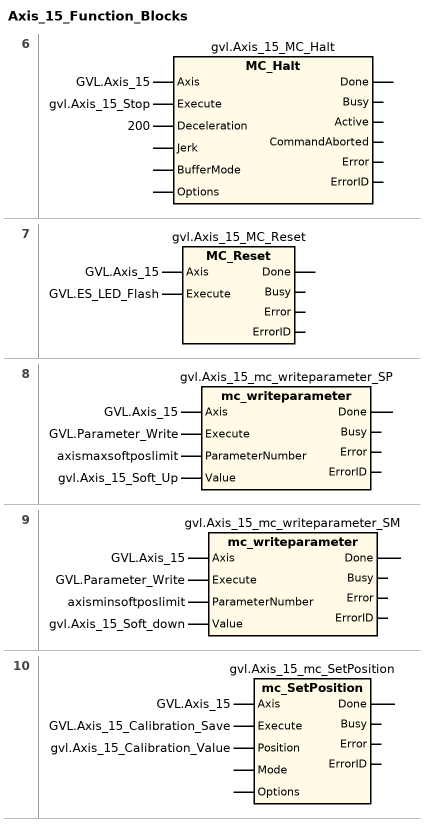
// NETWORK 6
gvl.Axis_15_MC_Halt(Axis := GVL.Axis_15, Execute := gvl.Axis_15_Stop, Deceleration := 200); // MC_Halt

// NETWORK 7
gvl.Axis_15_MC_Reset(Axis := GVL.Axis_15, Execute := GVL.ES_LED_Flash); // MC_Reset

// NETWORK 8
gvl.Axis_15_mc_writeparameter_SP(
    Axis := GVL.Axis_15,
    Execute := GVL.Parameter_Write,
    ParameterNumber := axismaxsoftposlimit,
    Value := gvl.Axis_15_Soft_Up); // mc_writeparameter

// NETWORK 9
gvl.Axis_15_mc_writeparameter_SM(
    Axis := GVL.Axis_15,
    Execute := GVL.Parameter_Write,
    ParameterNumber := axisminsoftposlimit,
    Value := gvl.Axis_15_Soft_down); // mc_writeparameter

// NETWORK 10
gvl.Axis_15_mc_SetPosition(
    Axis := GVL.Axis_15,
    Execute := GVL.Axis_15_Calibration_Save,
    Position := gvl.Axis_15_Calibration_Value); // mc_SetPosition

END_PROGRAM

// ---- POUs/Axis_15_Logic.TcPOU
PROGRAM Axis_15_Logic
VAR
	TON_0: TON;
	TON_1: TON;
	TON_2: TON;
	TON_3: TON;
	Axis_15_Velocity_Range: LREAL;
	Axis_15_Velocity_Scale: LREAL;
	Axis_15_Velocity_Raw: LREAL;
	Axis_15_Soft_Range: LREAL;
	Axis_15_Soft_Position: LREAL;
	Axis_15_Soft_Position_In_Range: LREAL;
END_VAR

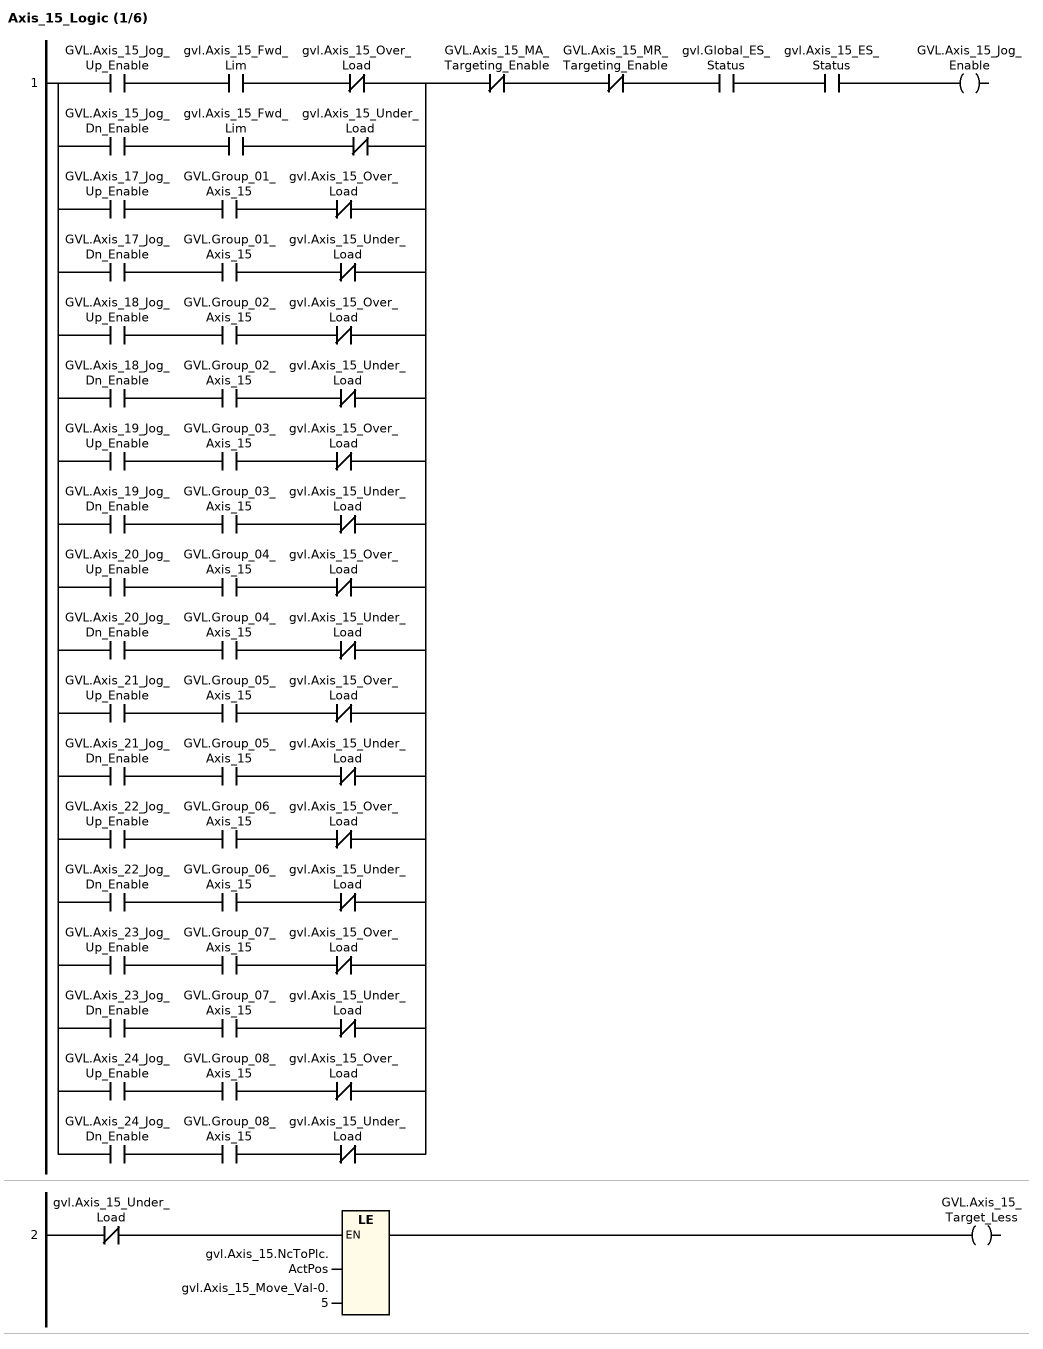
// NETWORK 1
GVL.Axis_15_Jog_Enable := (GVL.Axis_15_Jog_Up_Enable AND gvl.Axis_15_Fwd_Lim AND NOT gvl.Axis_15_Over_Load OR GVL.Axis_15_Jog_Dn_Enable AND gvl.Axis_15_Fwd_Lim AND NOT gvl.Axis_15_Under_Load OR GVL.Axis_17_Jog_Up_Enable AND GVL.Group_01_Axis_15 AND NOT gvl.Axis_15_Over_Load OR GVL.Axis_17_Jog_Dn_Enable AND GVL.Group_01_Axis_15 AND NOT gvl.Axis_15_Under_Load OR GVL.Axis_18_Jog_Up_Enable AND GVL.Group_02_Axis_15 AND NOT gvl.Axis_15_Over_Load OR GVL.Axis_18_Jog_Dn_Enable AND GVL.Group_02_Axis_15 AND NOT gvl.Axis_15_Under_Load OR GVL.Axis_19_Jog_Up_Enable AND GVL.Group_03_Axis_15 AND NOT gvl.Axis_15_Over_Load OR GVL.Axis_19_Jog_Dn_Enable AND GVL.Group_03_Axis_15 AND NOT gvl.Axis_15_Under_Load OR GVL.Axis_20_Jog_Up_Enable AND GVL.Group_04_Axis_15 AND NOT gvl.Axis_15_Over_Load OR GVL.Axis_20_Jog_Dn_Enable AND GVL.Group_04_Axis_15 AND NOT gvl.Axis_15_Under_Load OR GVL.Axis_21_Jog_Up_Enable AND GVL.Group_05_Axis_15 AND NOT gvl.Axis_15_Over_Load OR GVL.Axis_21_Jog_Dn_Enable AND GVL.Group_05_Axis_15 AND NOT gvl.Axis_15_Under_Load OR GVL.Axis_22_Jog_Up_Enable AND GVL.Group_06_Axis_15 AND NOT gvl.Axis_15_Over_Load OR GVL.Axis_22_Jog_Dn_Enable AND GVL.Group_06_Axis_15 AND NOT gvl.Axis_15_Under_Load OR GVL.Axis_23_Jog_Up_Enable AND GVL.Group_07_Axis_15 AND NOT gvl.Axis_15_Over_Load OR GVL.Axis_23_Jog_Dn_Enable AND GVL.Group_07_Axis_15 AND NOT gvl.Axis_15_Under_Load OR GVL.Axis_24_Jog_Up_Enable AND GVL.Group_08_Axis_15 AND NOT gvl.Axis_15_Over_Load OR GVL.Axis_24_Jog_Dn_Enable AND GVL.Group_08_Axis_15 AND NOT gvl.Axis_15_Under_Load) AND NOT GVL.Axis_15_MA_Targeting_Enable AND NOT GVL.Axis_15_MR_Targeting_Enable AND gvl.Global_ES_Status AND gvl.Axis_15_ES_Status;

// NETWORK 2
GVL.Axis_15_Target_Less := NOT gvl.Axis_15_Under_Load AND gvl.Axis_15.NcToPlc.ActPos <= (gvl.Axis_15_Move_Val-0.5);

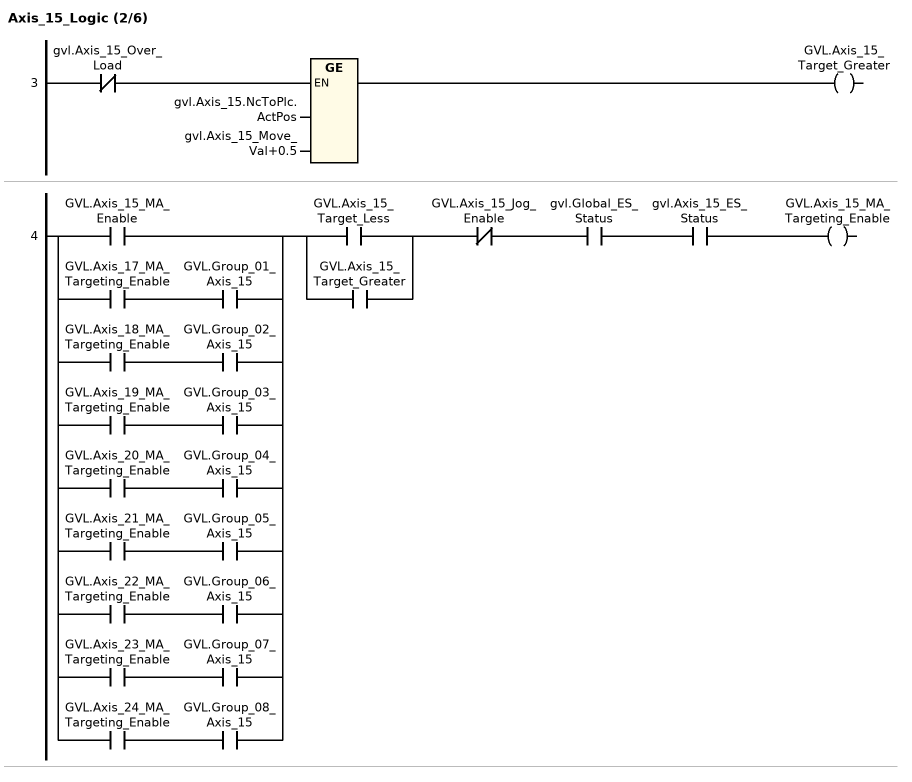
// NETWORK 3
GVL.Axis_15_Target_Greater := NOT gvl.Axis_15_Over_Load AND gvl.Axis_15.NcToPlc.ActPos >= (gvl.Axis_15_Move_Val+0.5);

// NETWORK 4
GVL.Axis_15_MA_Targeting_Enable := (GVL.Axis_15_MA_Enable OR GVL.Axis_17_MA_Targeting_Enable AND GVL.Group_01_Axis_15 OR GVL.Axis_18_MA_Targeting_Enable AND GVL.Group_02_Axis_15 OR GVL.Axis_19_MA_Targeting_Enable AND GVL.Group_03_Axis_15 OR GVL.Axis_20_MA_Targeting_Enable AND GVL.Group_04_Axis_15 OR GVL.Axis_21_MA_Targeting_Enable AND GVL.Group_05_Axis_15 OR GVL.Axis_22_MA_Targeting_Enable AND GVL.Group_06_Axis_15 OR GVL.Axis_23_MA_Targeting_Enable AND GVL.Group_07_Axis_15 OR GVL.Axis_24_MA_Targeting_Enable AND GVL.Group_08_Axis_15) AND (GVL.Axis_15_Target_Less OR GVL.Axis_15_Target_Greater) AND NOT GVL.Axis_15_Jog_Enable AND gvl.Global_ES_Status AND gvl.Axis_15_ES_Status;

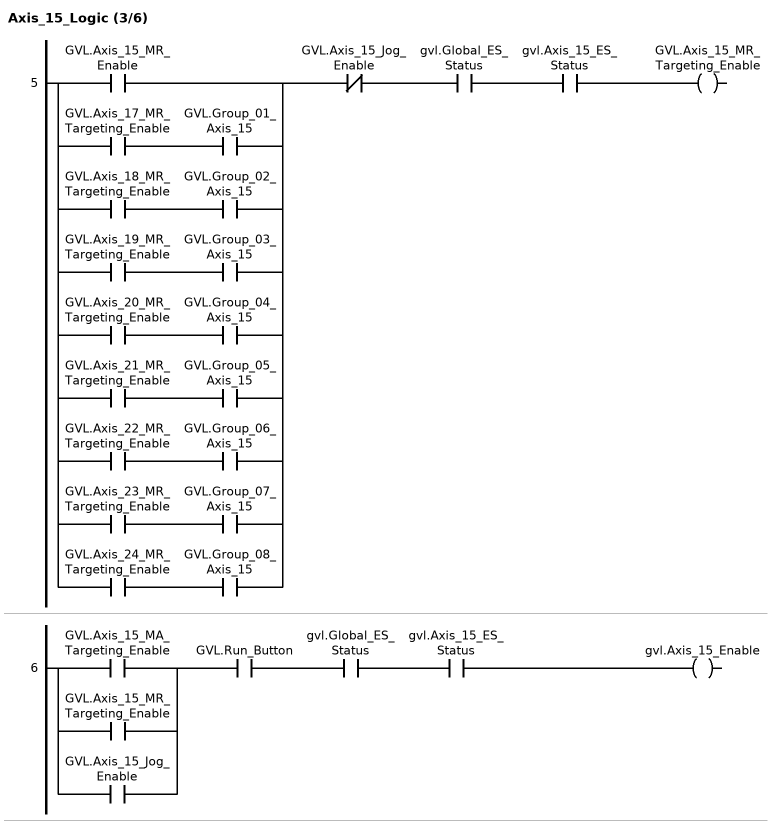
// NETWORK 5
GVL.Axis_15_MR_Targeting_Enable := (GVL.Axis_15_MR_Enable OR GVL.Axis_17_MR_Targeting_Enable AND GVL.Group_01_Axis_15 OR GVL.Axis_18_MR_Targeting_Enable AND GVL.Group_02_Axis_15 OR GVL.Axis_19_MR_Targeting_Enable AND GVL.Group_03_Axis_15 OR GVL.Axis_20_MR_Targeting_Enable AND GVL.Group_04_Axis_15 OR GVL.Axis_21_MR_Targeting_Enable AND GVL.Group_05_Axis_15 OR GVL.Axis_22_MR_Targeting_Enable AND GVL.Group_06_Axis_15 OR GVL.Axis_23_MR_Targeting_Enable AND GVL.Group_07_Axis_15 OR GVL.Axis_24_MR_Targeting_Enable AND GVL.Group_08_Axis_15) AND NOT GVL.Axis_15_Jog_Enable AND gvl.Global_ES_Status AND gvl.Axis_15_ES_Status;

// NETWORK 6
gvl.Axis_15_Enable := (GVL.Axis_15_MA_Targeting_Enable OR GVL.Axis_15_MR_Targeting_Enable OR GVL.Axis_15_Jog_Enable) AND GVL.Run_Button AND gvl.Global_ES_Status AND gvl.Axis_15_ES_Status;

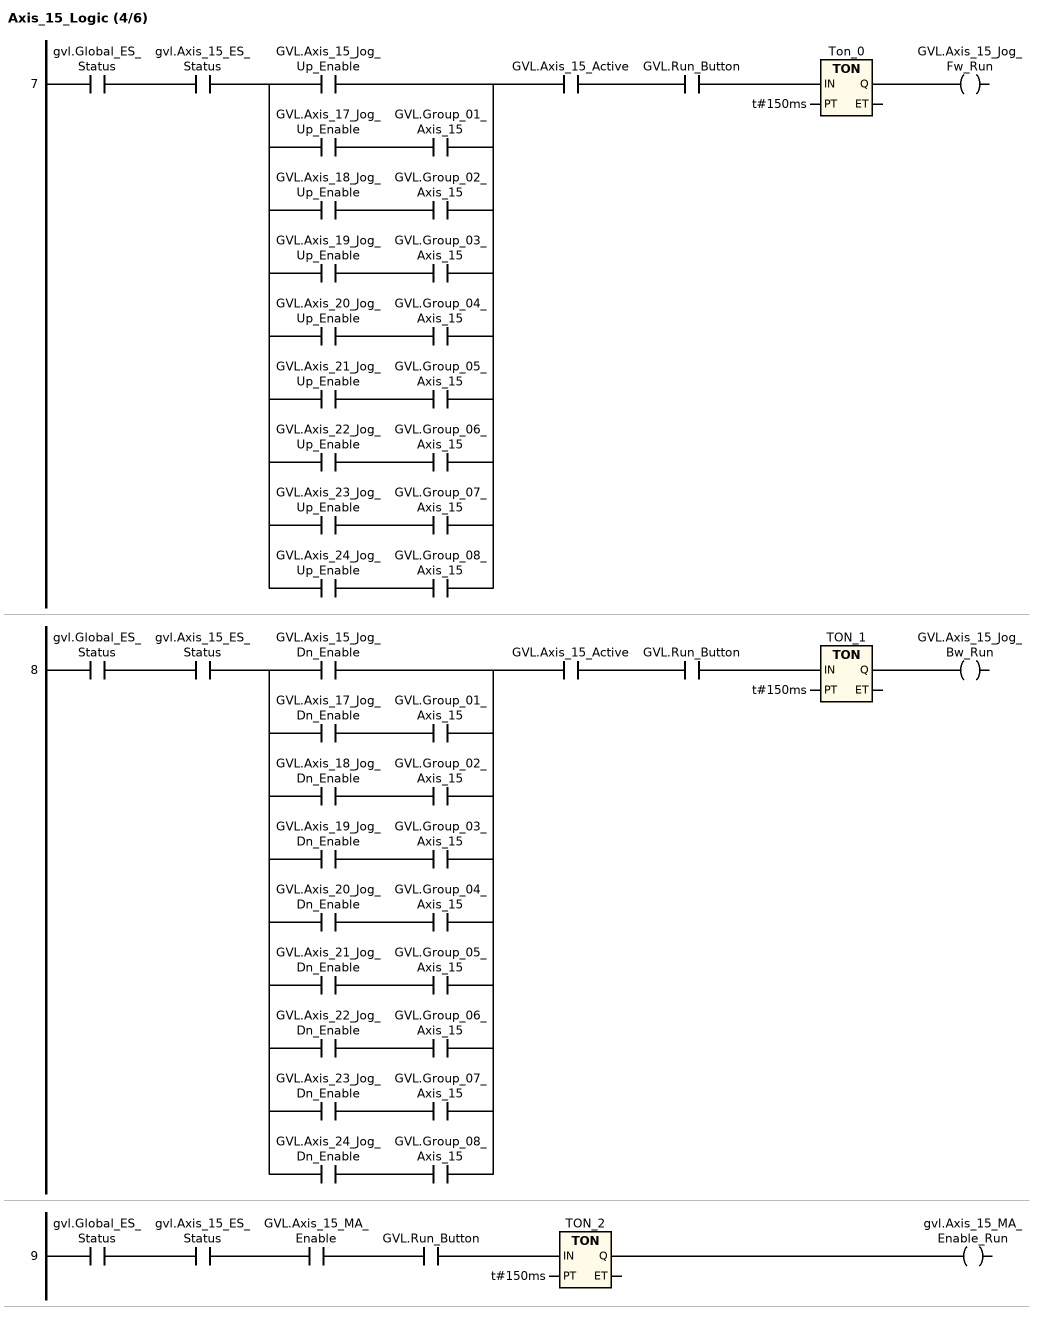
// NETWORK 7
Ton_0(IN := gvl.Global_ES_Status AND gvl.Axis_15_ES_Status AND (GVL.Axis_15_Jog_Up_Enable OR GVL.Axis_17_Jog_Up_Enable AND GVL.Group_01_Axis_15 OR GVL.Axis_18_Jog_Up_Enable AND GVL.Group_02_Axis_15 OR GVL.Axis_19_Jog_Up_Enable AND GVL.Group_03_Axis_15 OR GVL.Axis_20_Jog_Up_Enable AND GVL.Group_04_Axis_15 OR GVL.Axis_21_Jog_Up_Enable AND GVL.Group_05_Axis_15 OR GVL.Axis_22_Jog_Up_Enable AND GVL.Group_06_Axis_15 OR GVL.Axis_23_Jog_Up_Enable AND GVL.Group_07_Axis_15 OR GVL.Axis_24_Jog_Up_Enable AND GVL.Group_08_Axis_15) AND GVL.Axis_15_Active AND GVL.Run_Button, PT := t#150ms); // TON
GVL.Axis_15_Jog_Fw_Run := Ton_0.Q;

// NETWORK 8
TON_1(IN := gvl.Global_ES_Status AND gvl.Axis_15_ES_Status AND (GVL.Axis_15_Jog_Dn_Enable OR GVL.Axis_17_Jog_Dn_Enable AND GVL.Group_01_Axis_15 OR GVL.Axis_18_Jog_Dn_Enable AND GVL.Group_02_Axis_15 OR GVL.Axis_19_Jog_Dn_Enable AND GVL.Group_03_Axis_15 OR GVL.Axis_20_Jog_Dn_Enable AND GVL.Group_04_Axis_15 OR GVL.Axis_21_Jog_Dn_Enable AND GVL.Group_05_Axis_15 OR GVL.Axis_22_Jog_Dn_Enable AND GVL.Group_06_Axis_15 OR GVL.Axis_23_Jog_Dn_Enable AND GVL.Group_07_Axis_15 OR GVL.Axis_24_Jog_Dn_Enable AND GVL.Group_08_Axis_15) AND GVL.Axis_15_Active AND GVL.Run_Button, PT := t#150ms); // TON
GVL.Axis_15_Jog_Bw_Run := TON_1.Q;

// NETWORK 9
TON_2(IN := gvl.Global_ES_Status AND gvl.Axis_15_ES_Status AND GVL.Axis_15_MA_Enable AND GVL.Run_Button, PT := t#150ms); // TON
gvl.Axis_15_MA_Enable_Run := TON_2.Q;

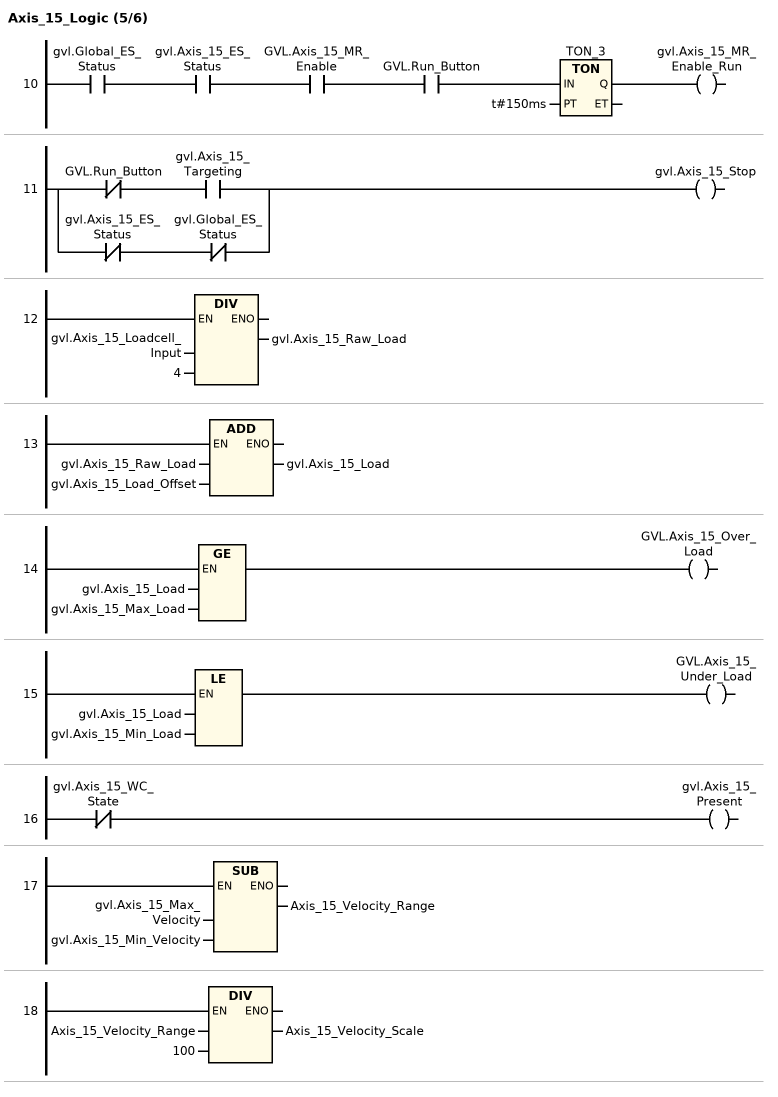
// NETWORK 10
TON_3(IN := gvl.Global_ES_Status AND gvl.Axis_15_ES_Status AND GVL.Axis_15_MR_Enable AND GVL.Run_Button, PT := t#150ms); // TON
gvl.Axis_15_MR_Enable_Run := TON_3.Q;

// NETWORK 11
gvl.Axis_15_Stop := NOT GVL.Run_Button AND gvl.Axis_15_Targeting OR NOT gvl.Axis_15_ES_Status AND NOT gvl.Global_ES_Status;

// NETWORK 12
gvl.Axis_15_Raw_Load := gvl.Axis_15_Loadcell_Input / 4;

// NETWORK 13
gvl.Axis_15_Load := gvl.Axis_15_Raw_Load + gvl.Axis_15_Load_Offset;

// NETWORK 14
GVL.Axis_15_Over_Load := gvl.Axis_15_Load >= gvl.Axis_15_Max_Load;

// NETWORK 15
GVL.Axis_15_Under_Load := gvl.Axis_15_Load <= gvl.Axis_15_Min_Load;

// NETWORK 16
gvl.Axis_15_Present := NOT gvl.Axis_15_WC_State;

// NETWORK 17
Axis_15_Velocity_Range := gvl.Axis_15_Max_Velocity - gvl.Axis_15_Min_Velocity;

// NETWORK 18
Axis_15_Velocity_Scale := Axis_15_Velocity_Range / 100;

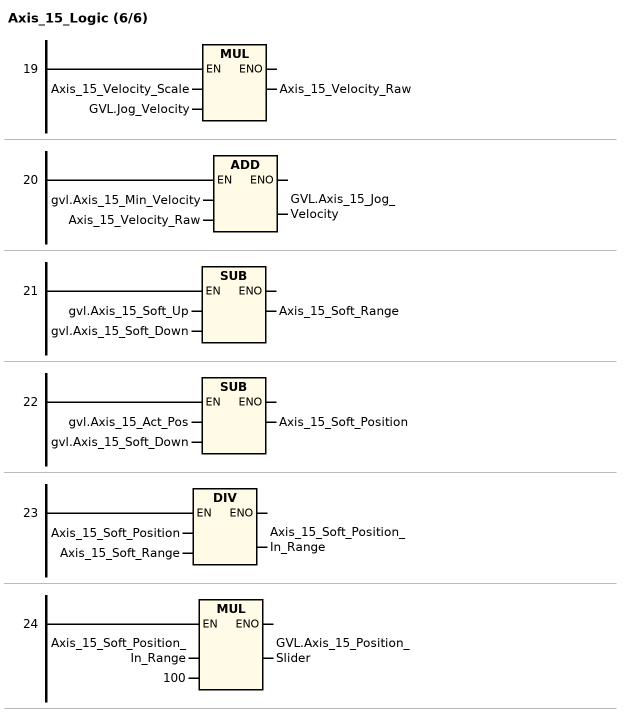
// NETWORK 19
Axis_15_Velocity_Raw := Axis_15_Velocity_Scale * GVL.Jog_Velocity;

// NETWORK 20
GVL.Axis_15_Jog_Velocity := gvl.Axis_15_Min_Velocity + Axis_15_Velocity_Raw;

// NETWORK 21
Axis_15_Soft_Range := gvl.Axis_15_Soft_Up - gvl.Axis_15_Soft_Down;

// NETWORK 22
Axis_15_Soft_Position := gvl.Axis_15_Act_Pos - gvl.Axis_15_Soft_Down;

// NETWORK 23
Axis_15_Soft_Position_In_Range := Axis_15_Soft_Position / Axis_15_Soft_Range;

// NETWORK 24
GVL.Axis_15_Position_Slider := Axis_15_Soft_Position_In_Range * 100;

END_PROGRAM

// ---- POUs/Axis_16_Function_Blocks.TcPOU
PROGRAM Axis_16_Function_Blocks
VAR
END_VAR

